TYPE ST_Powerstack_Service :
STRUCT
	Netcontactor			: St_Netcontactor_service;
	PowermoduleMaster		: ST_Powermodule_Service;
	PowermoduleSlave		: ST_Powermodule_Service;
END_STRUCT
END_TYPE

(* stored: Version 1.1.0.1, ProductVersion 3.1.4026.18
   DUT ST_Powerstack_Service: Id {b7261a14-bcc5-49f5-abb8-762990946357} *)
